(* Logix 5000 project; controller cal1615 1756-L62 rev 20.11; software revision 20.05; part 19 of 81 *)
(* tags used below, declared in another part *)
   FAULT : BOOL;   // Fault AFI
   HMI : BOOL;   // AFI HMI
   p01_param_oven_timer_presets : DINT[32];   // System Parameter Oven Timer Presets
   p01_param_process_air_hl : REAL;   // Machine Parameter Process Air High Limit
   p01_sys_lc : Limit_Clamp;   // Zone 1 Misc Control Limit Clamp
   p01r09_pb_global_reset : BOOL;   // System Modes PB: Global Fault Reset
   p01r11 : routine;   // System Timer Presets
   p02_real_from_hmi : hmi_real;   // MOP HMI Iface Real from HMI
   p11_dint_to_hmi : DINT[16];   // Zone 1 Temperature Control VFDs On
   p11_param_fast_to_soak : REAL;   // Zone 1 Parameter Fast to Soak Control
   p11_param_lfl_hhl : REAL;   // Zone 1 Parameter High High Lower Flash Limit
   p11_param_lfl_hl : REAL;   // Zone 1 Parameter High LFL Limit
   p11_param_pid1_ff : REAL;   // Zone 1 Parameter Fast PID Bias
   p11_param_pid1_kd : REAL;   // Zone 1 Parameter Fast PID Derivative Gain
   p11_param_pid1_ki : REAL;   // Zone 1 Parameter Fast PID Integral Gain
   p11_param_pid1_kp : REAL;   // Zone 1 Parameter Fast PID Proportional Gain
   p11_param_pid2_ff : REAL;   // Zone 1 Parameter Auto PID Bias
   p11_param_pid2_kd : REAL;   // Zone 1 Parameter Auto PID Derivative Gain
   p11_param_pid2_ki : REAL;   // Zone 1 Parameter Auto PID Integral Gain
   p11_param_pid2_kp : REAL;   // Zone 1 Parameter Auto PID Proportional Gain
   p11_param_shutdown_temp : REAL;   // Zone 1 Parameter Zone Shutdown Temperature
   p11_param_soak_to_fast : REAL;   // Zone 1 Parameter Soak to Fast Control
   p11_param_tc01_dev : REAL;   // Zone 1 Parameter Oven Temperature Deviation from Setpoint
   p11_param_tc01_hl : REAL;   // Zone 1 Parameter Process Air High Limit
   p11_param_tc01z : REAL;   // Zone 1 Parameter Process Temperature Zero Offset
   p11_param_tc02z : REAL;   // Zone 1 Parameter SupplyTemperature Zero Offset
   p11_param_zone_pressure : REAL;   // Zone 1 Parameter High Pressure LImit
   p11r01 : routine;   // Zone 1 Main
   p11r02 : routine;   // Zone 1 Misc Control
   p11r02_timer_warning : TIMER[4];   // Zone 1 Misc Control Warning Delay
   p11r07 : routine;   // Zone 1 Alarms
   p11r07_timer_fault : TIMER[4];   // Zone 1 Alarms Fault Delay
   p11r07_timer_warning : TIMER[4];   // Zone 1 Alarms Warning Delay
   p11r08 : routine;   // Zone 1 Warnings
   p11r08_timer_fault : TIMER[4];   // Zone 1 Warnings Fault Delay
   p11r08_timer_warning : TIMER[4];   // Zone 1 Warnings Warning Delay
   p11r09 : routine;   // Zone 1 Modes
   p11r09_timer_fault : TIMER[4];   // Zone 1 Modes Fault Delay
   p11r09_timer_warning : TIMER[8];   // Zone 1 Modes Warning Delay
   p11r10 : routine;   // Zone 1
   p11r20 : routine;   // Zone 1 Temp Sequence
   p11r30 : routine;   // Zone 1 Temperature Control
   p11r30_cv_man_sp : REAL;   // Zone 1 Temperature Control Manual Heat Control Valve Setpoint
   p11r30_temp_deviation_setpoint : DINT;
   p11r30_timer_fault : TIMER[16];   // Zone 1 Temperature Control Fault Delay
   p11r30_timer_warning : TIMER[12];   // Zone 1 Temperature Control Warning Delay
   p11r31 : routine;   // Zone 1 Exhaust VFD
   p11r31_timer_fault : TIMER[5];   // Zone 1 Exhaust VFD Fault Timer
   p11r31_timer_warning : TIMER[5];   // Zone 1 Exhaust VFD Waringing Timer
   p11r32 : routine;   // Zone 1 Recirc VFD
   p11r32_timer_fault : TIMER[5];   // Zone 1 Recirc VFD Fault Timer
   p11r32_timer_warning : TIMER[5];   // Zone 1 Supply VFD Warning Timer
(* P11_Zone_1, continued *)

ROUTINE R07_Alarms   (* ladder *)
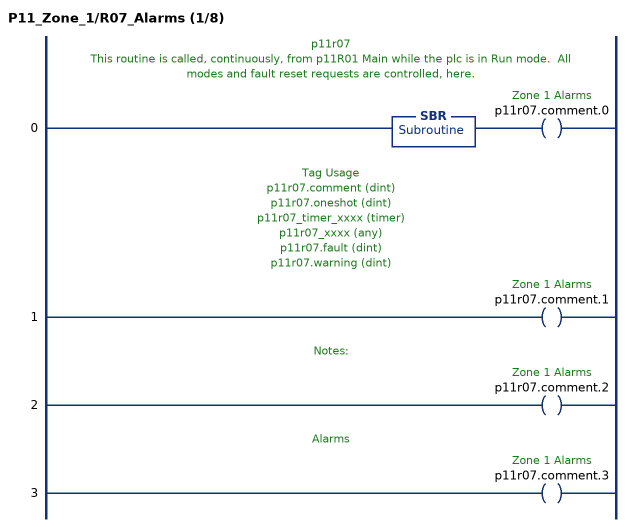
   // p11r07
   // This routine is called, continuously, from p11R01 Main while the plc is in Run mode.  All modes and fault reset requests are controlled, here.
   0: SBR()OTE(p11r07.comment.0);
   // Tag Usage
   // p11r07.comment (dint)
   // p11r07.oneshot (dint)
   // p11r07_timer_xxxx (timer)
   // p11r07_xxxx (any)
   // p11r07.fault (dint)
   // p11r07.warning (dint)
   1: OTE(p11r07.comment.1);
   // Notes:
   2: OTE(p11r07.comment.2);
   // Alarms
   3: OTE(p11r07.comment.3);
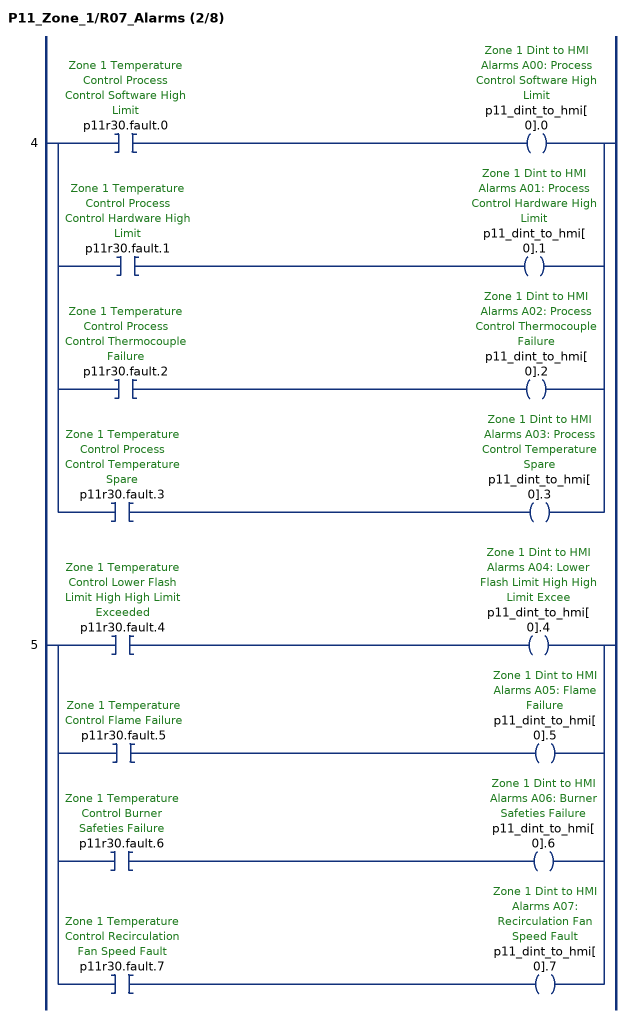
   4: [XIC(p11r30.fault.0) OTE(p11_dint_to_hmi[0].0) ,XIC(p11r30.fault.1) OTE(p11_dint_to_hmi[0].1) ,XIC(p11r30.fault.2) OTE(p11_dint_to_hmi[0].2) ,XIC(p11r30.fault.3) OTE(p11_dint_to_hmi[0].3) ];
   5: [XIC(p11r30.fault.4) OTE(p11_dint_to_hmi[0].4) ,XIC(p11r30.fault.5) OTE(p11_dint_to_hmi[0].5) ,XIC(p11r30.fault.6) OTE(p11_dint_to_hmi[0].6) ,XIC(p11r30.fault.7) OTE(p11_dint_to_hmi[0].7) ];
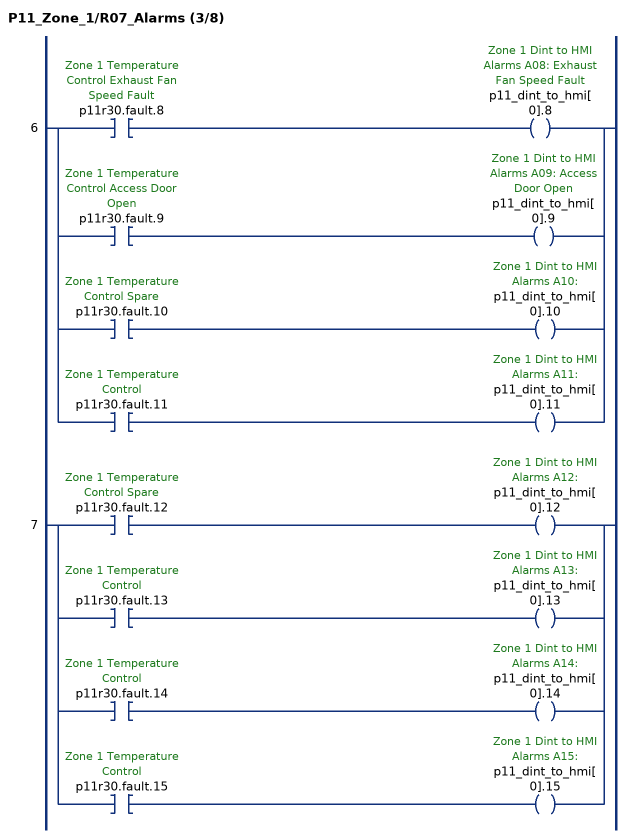
   6: [XIC(p11r30.fault.8) OTE(p11_dint_to_hmi[0].8) ,XIC(p11r30.fault.9) OTE(p11_dint_to_hmi[0].9) ,XIC(p11r30.fault.10) OTE(p11_dint_to_hmi[0].10) ,XIC(p11r30.fault.11) OTE(p11_dint_to_hmi[0].11) ];
   7: [XIC(p11r30.fault.12) OTE(p11_dint_to_hmi[0].12) ,XIC(p11r30.fault.13) OTE(p11_dint_to_hmi[0].13) ,XIC(p11r30.fault.14) OTE(p11_dint_to_hmi[0].14) ,XIC(p11r30.fault.15) OTE(p11_dint_to_hmi[0].15) ];
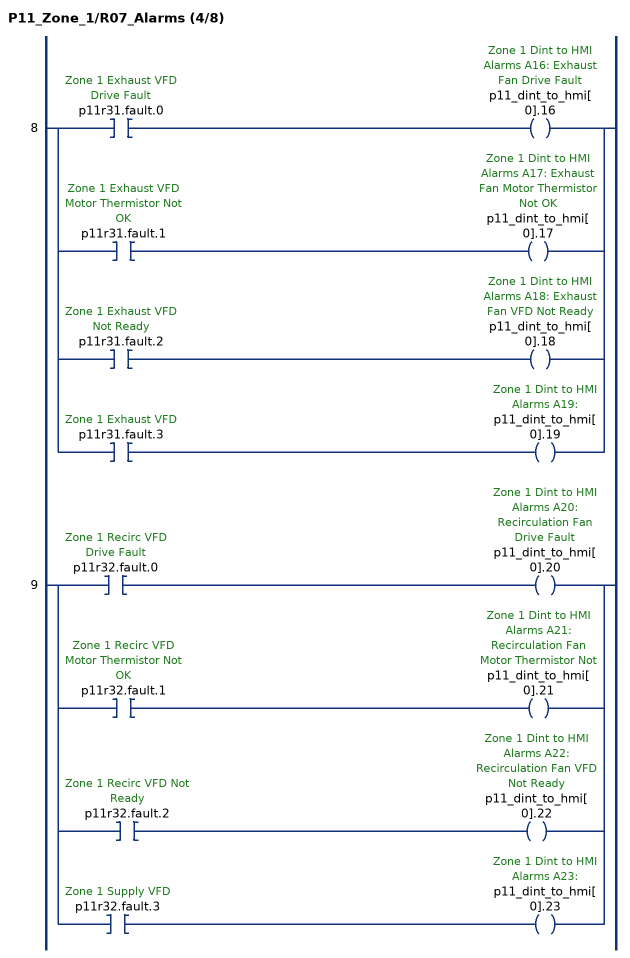
   8: [XIC(p11r31.fault.0) OTE(p11_dint_to_hmi[0].16) ,XIC(p11r31.fault.1) OTE(p11_dint_to_hmi[0].17) ,XIC(p11r31.fault.2) OTE(p11_dint_to_hmi[0].18) ,XIC(p11r31.fault.3) OTE(p11_dint_to_hmi[0].19) ];
   9: [XIC(p11r32.fault.0) OTE(p11_dint_to_hmi[0].20) ,XIC(p11r32.fault.1) OTE(p11_dint_to_hmi[0].21) ,XIC(p11r32.fault.2) OTE(p11_dint_to_hmi[0].22) ,XIC(p11r32.fault.3) OTE(p11_dint_to_hmi[0].23) ];
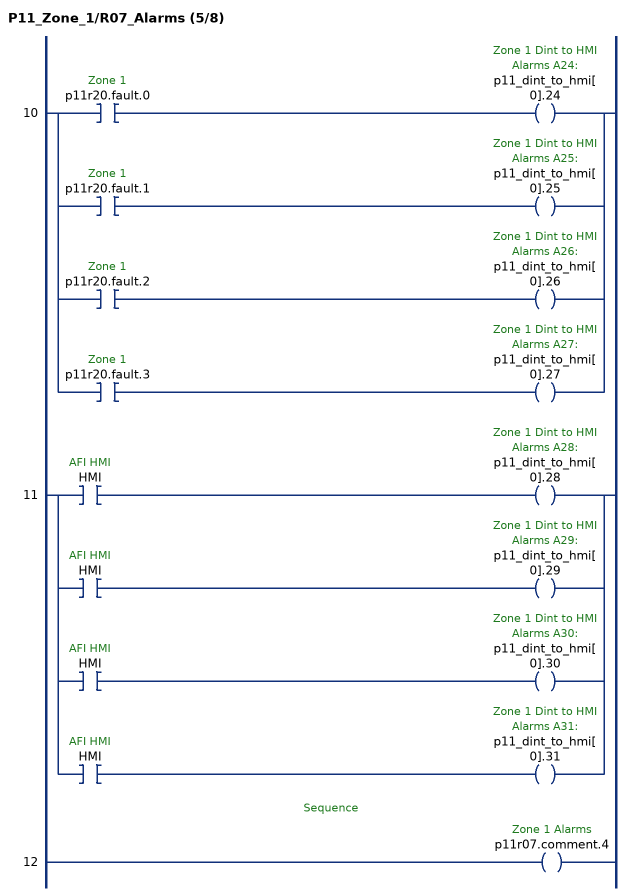
   10: [XIC(p11r20.fault.0) OTE(p11_dint_to_hmi[0].24) ,XIC(p11r20.fault.1) OTE(p11_dint_to_hmi[0].25) ,XIC(p11r20.fault.2) OTE(p11_dint_to_hmi[0].26) ,XIC(p11r20.fault.3) OTE(p11_dint_to_hmi[0].27) ];
   11: [XIC(HMI) OTE(p11_dint_to_hmi[0].28) ,XIC(HMI) OTE(p11_dint_to_hmi[0].29) ,XIC(HMI) OTE(p11_dint_to_hmi[0].30) ,XIC(HMI) OTE(p11_dint_to_hmi[0].31) ];
   // Sequence
   12: OTE(p11r07.comment.4);
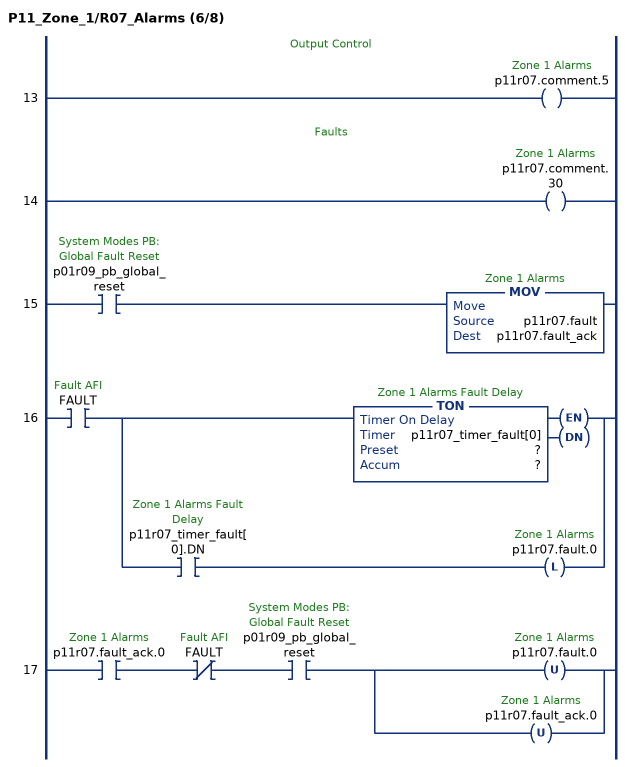
   // Output Control
   13: OTE(p11r07.comment.5);
   // Faults
   14: OTE(p11r07.comment.30);
   15: XIC(p01r09_pb_global_reset)MOV(p11r07.fault,p11r07.fault_ack);
   16: XIC(FAULT)[TON(p11r07_timer_fault[0],?,?) ,XIC(p11r07_timer_fault[0].DN) OTL(p11r07.fault.0) ];
   17: XIC(p11r07.fault_ack.0)XIO(FAULT)XIC(p01r09_pb_global_reset)[OTU(p11r07.fault.0) ,OTU(p11r07.fault_ack.0) ];
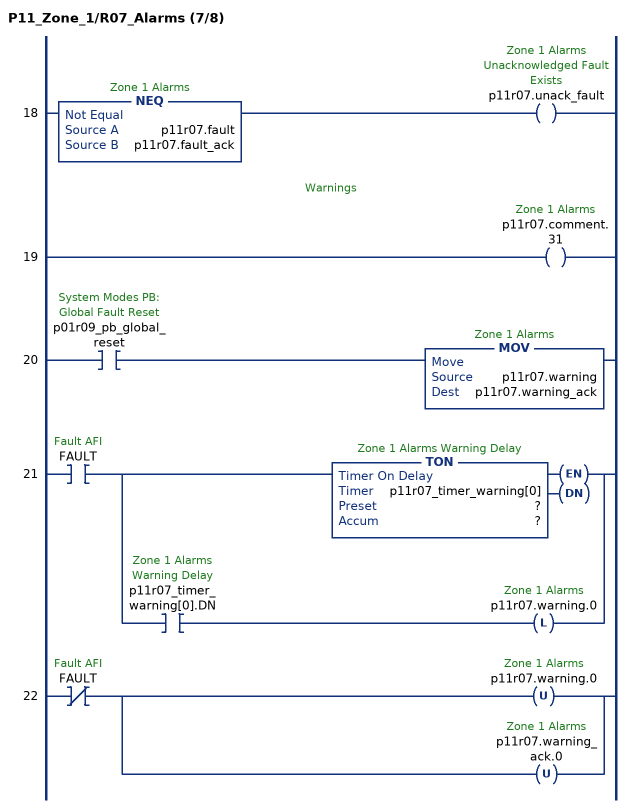
   18: NEQ(p11r07.fault,p11r07.fault_ack)OTE(p11r07.unack_fault);
   // Warnings
   19: OTE(p11r07.comment.31);
   20: XIC(p01r09_pb_global_reset)MOV(p11r07.warning,p11r07.warning_ack);
   21: XIC(FAULT)[TON(p11r07_timer_warning[0],?,?) ,XIC(p11r07_timer_warning[0].DN) OTL(p11r07.warning.0) ];
   22: XIO(FAULT)[OTU(p11r07.warning.0) ,OTU(p11r07.warning_ack.0) ];
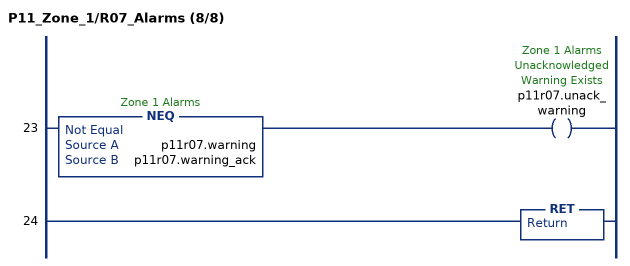
   23: NEQ(p11r07.warning,p11r07.warning_ack)OTE(p11r07.unack_warning);
   24: RET();
END_ROUTINE

ROUTINE R08_Warnings   (* ladder *)
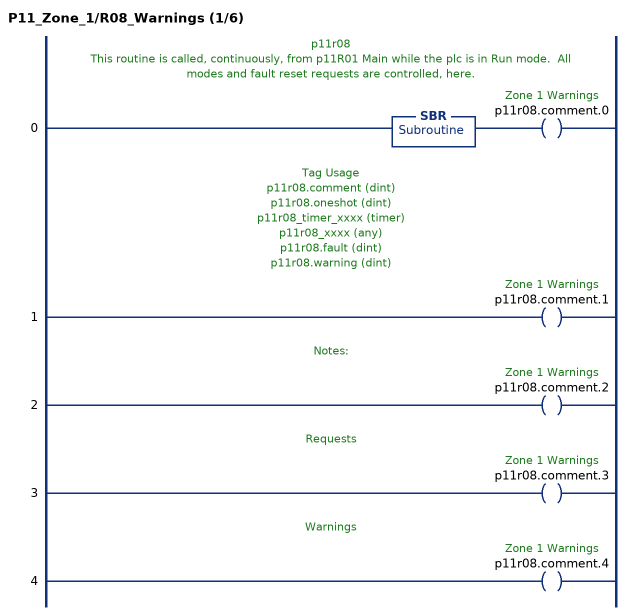
   // p11r08
   // This routine is called, continuously, from p11R01 Main while the plc is in Run mode.  All modes and fault reset requests are controlled, here.
   0: SBR()OTE(p11r08.comment.0);
   // Tag Usage
   // p11r08.comment (dint)
   // p11r08.oneshot (dint)
   // p11r08_timer_xxxx (timer)
   // p11r08_xxxx (any)
   // p11r08.fault (dint)
   // p11r08.warning (dint)
   1: OTE(p11r08.comment.1);
   // Notes:
   2: OTE(p11r08.comment.2);
   // Requests
   3: OTE(p11r08.comment.3);
   // Warnings
   4: OTE(p11r08.comment.4);
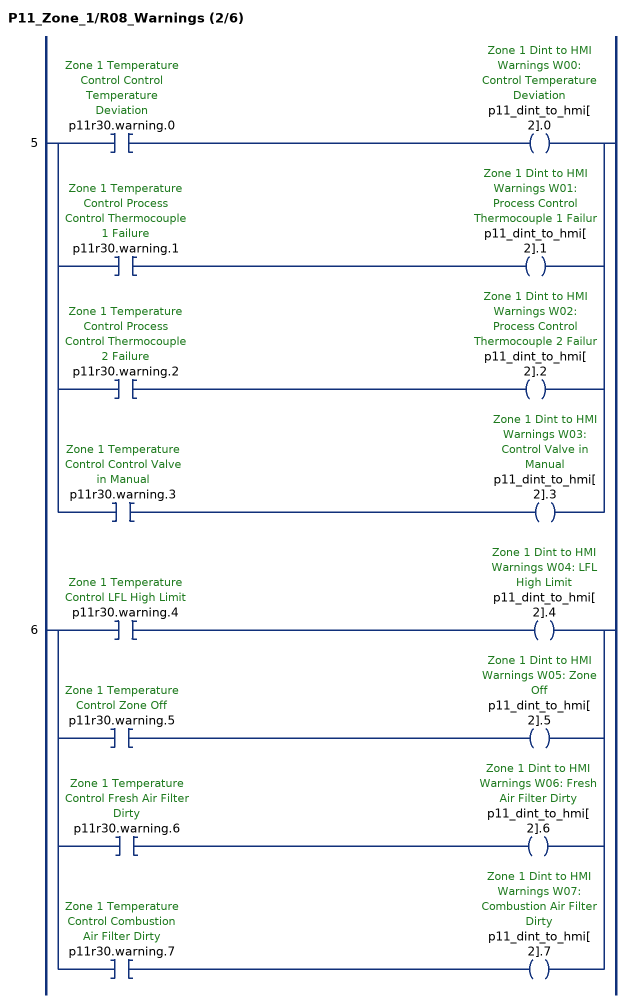
   5: [XIC(p11r30.warning.0) OTE(p11_dint_to_hmi[2].0) ,XIC(p11r30.warning.1) OTE(p11_dint_to_hmi[2].1) ,XIC(p11r30.warning.2) OTE(p11_dint_to_hmi[2].2) ,XIC(p11r30.warning.3) OTE(p11_dint_to_hmi[2].3) ];
   6: [XIC(p11r30.warning.4) OTE(p11_dint_to_hmi[2].4) ,XIC(p11r30.warning.5) OTE(p11_dint_to_hmi[2].5) ,XIC(p11r30.warning.6) OTE(p11_dint_to_hmi[2].6) ,XIC(p11r30.warning.7) OTE(p11_dint_to_hmi[2].7) ];
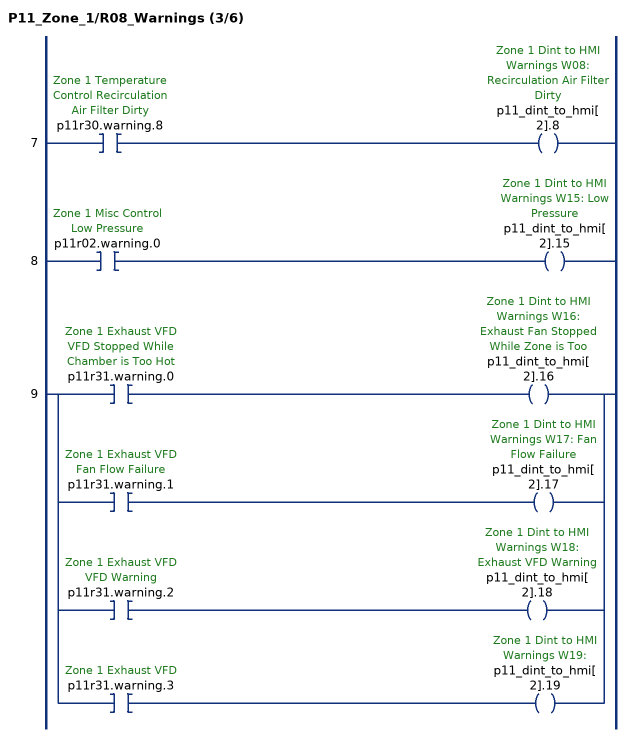
   7: XIC(p11r30.warning.8)OTE(p11_dint_to_hmi[2].8);
   8: XIC(p11r02.warning.0)OTE(p11_dint_to_hmi[2].15);
   9: [XIC(p11r31.warning.0) OTE(p11_dint_to_hmi[2].16) ,XIC(p11r31.warning.1) OTE(p11_dint_to_hmi[2].17) ,XIC(p11r31.warning.2) OTE(p11_dint_to_hmi[2].18) ,XIC(p11r31.warning.3) OTE(p11_dint_to_hmi[2].19) ];
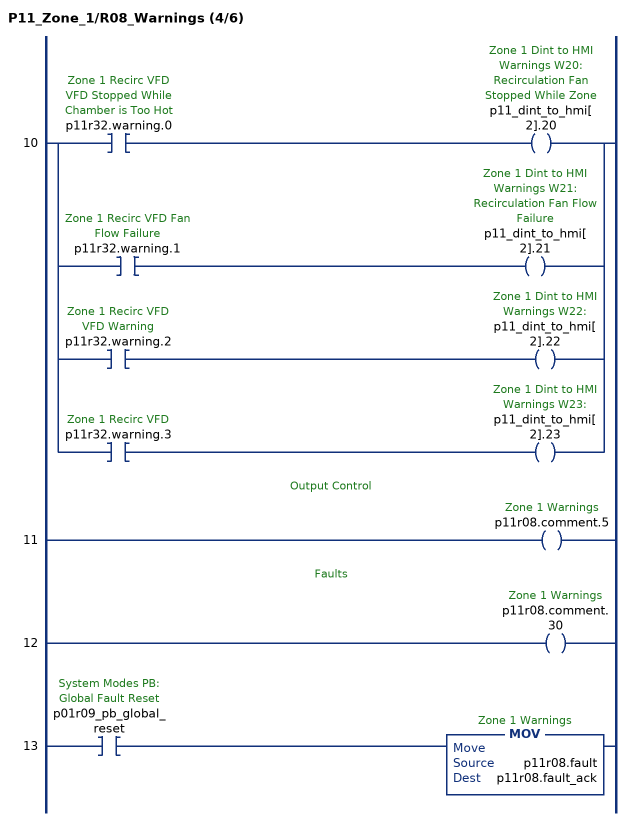
   10: [XIC(p11r32.warning.0) OTE(p11_dint_to_hmi[2].20) ,XIC(p11r32.warning.1) OTE(p11_dint_to_hmi[2].21) ,XIC(p11r32.warning.2) OTE(p11_dint_to_hmi[2].22) ,XIC(p11r32.warning.3) OTE(p11_dint_to_hmi[2].23) ];
   // Output Control
   11: OTE(p11r08.comment.5);
   // Faults
   12: OTE(p11r08.comment.30);
   13: XIC(p01r09_pb_global_reset)MOV(p11r08.fault,p11r08.fault_ack);
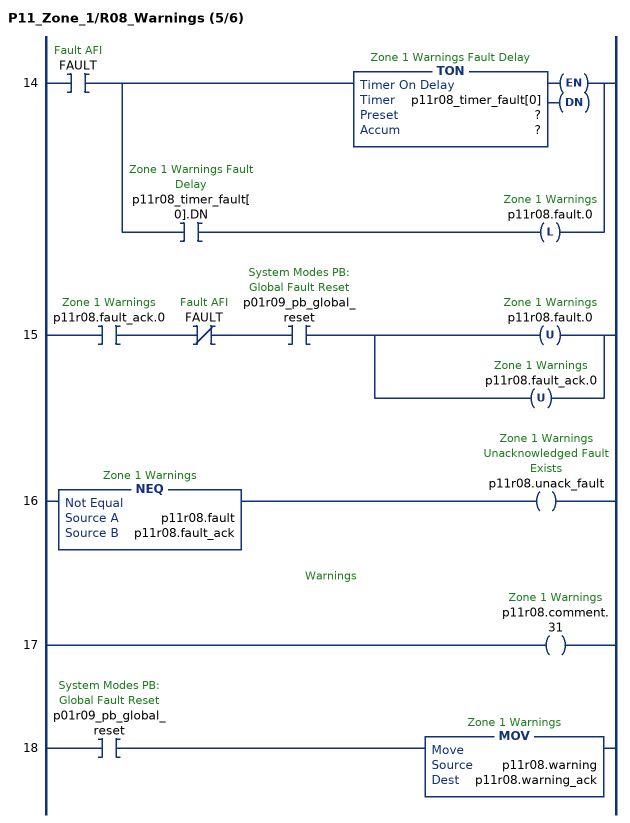
   14: XIC(FAULT)[TON(p11r08_timer_fault[0],?,?) ,XIC(p11r08_timer_fault[0].DN) OTL(p11r08.fault.0) ];
   15: XIC(p11r08.fault_ack.0)XIO(FAULT)XIC(p01r09_pb_global_reset)[OTU(p11r08.fault.0) ,OTU(p11r08.fault_ack.0) ];
   16: NEQ(p11r08.fault,p11r08.fault_ack)OTE(p11r08.unack_fault);
   // Warnings
   17: OTE(p11r08.comment.31);
   18: XIC(p01r09_pb_global_reset)MOV(p11r08.warning,p11r08.warning_ack);
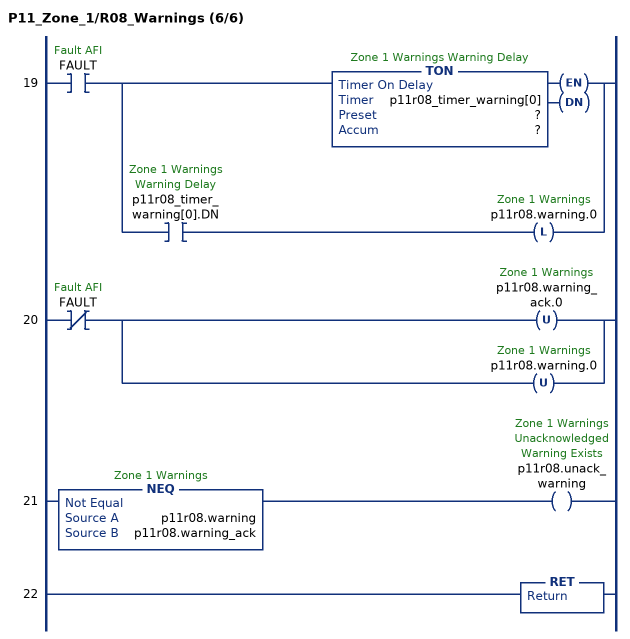
   19: XIC(FAULT)[TON(p11r08_timer_warning[0],?,?) ,XIC(p11r08_timer_warning[0].DN) OTL(p11r08.warning.0) ];
   20: XIO(FAULT)[OTU(p11r08.warning_ack.0) ,OTU(p11r08.warning.0) ];
   21: NEQ(p11r08.warning,p11r08.warning_ack)OTE(p11r08.unack_warning);
   22: RET();
END_ROUTINE

ROUTINE R09_Modes   (* ladder *)
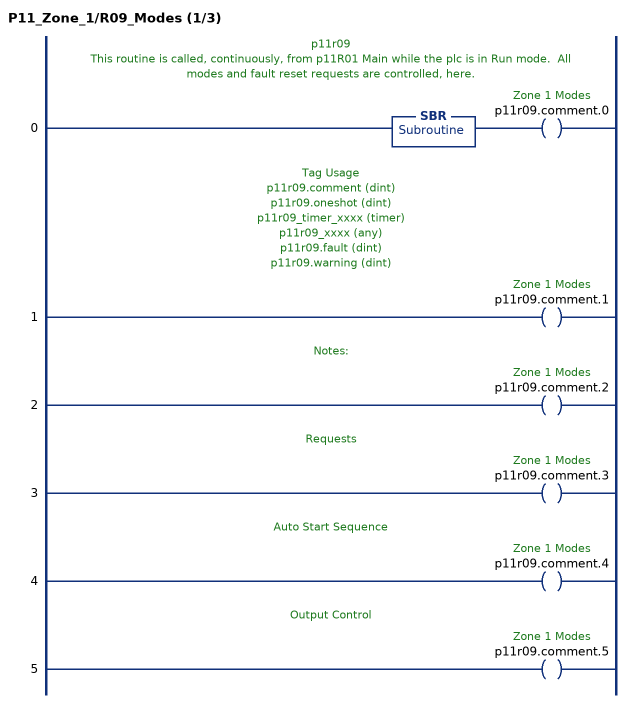
   // p11r09
   // This routine is called, continuously, from p11R01 Main while the plc is in Run mode.  All modes and fault reset requests are controlled, here.
   0: SBR()OTE(p11r09.comment.0);
   // Tag Usage
   // p11r09.comment (dint)
   // p11r09.oneshot (dint)
   // p11r09_timer_xxxx (timer)
   // p11r09_xxxx (any)
   // p11r09.fault (dint)
   // p11r09.warning (dint)
   1: OTE(p11r09.comment.1);
   // Notes:
   2: OTE(p11r09.comment.2);
   // Requests
   3: OTE(p11r09.comment.3);
   // Auto Start Sequence
   4: OTE(p11r09.comment.4);
   // Output Control
   5: OTE(p11r09.comment.5);
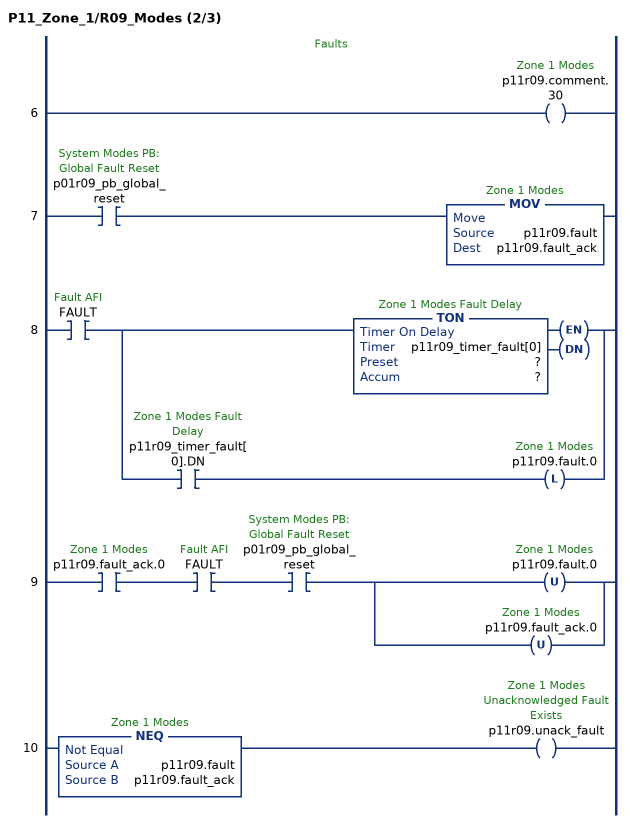
   // Faults
   6: OTE(p11r09.comment.30);
   7: XIC(p01r09_pb_global_reset)MOV(p11r09.fault,p11r09.fault_ack);
   8: XIC(FAULT)[TON(p11r09_timer_fault[0],?,?) ,XIC(p11r09_timer_fault[0].DN) OTL(p11r09.fault.0) ];
   9: XIC(p11r09.fault_ack.0)XIC(FAULT)XIC(p01r09_pb_global_reset)[OTU(p11r09.fault.0) ,OTU(p11r09.fault_ack.0) ];
   10: NEQ(p11r09.fault,p11r09.fault_ack)OTE(p11r09.unack_fault);
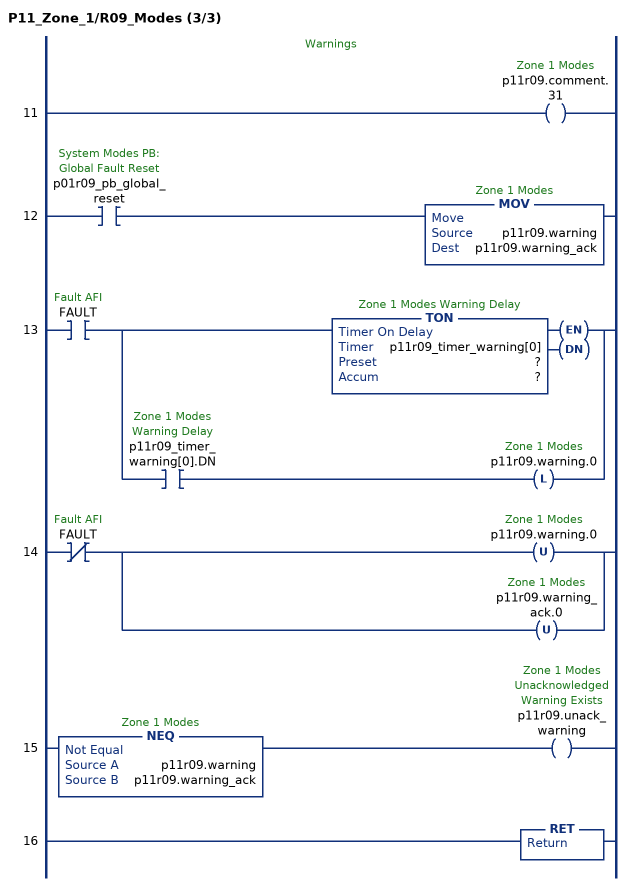
   // Warnings
   11: OTE(p11r09.comment.31);
   12: XIC(p01r09_pb_global_reset)MOV(p11r09.warning,p11r09.warning_ack);
   13: XIC(FAULT)[TON(p11r09_timer_warning[0],?,?) ,XIC(p11r09_timer_warning[0].DN) OTL(p11r09.warning.0) ];
   14: XIO(FAULT)[OTU(p11r09.warning.0) ,OTU(p11r09.warning_ack.0) ];
   15: NEQ(p11r09.warning,p11r09.warning_ack)OTE(p11r09.unack_warning);
   16: RET();
END_ROUTINE

ROUTINE R10_Parameters   (* ladder *)
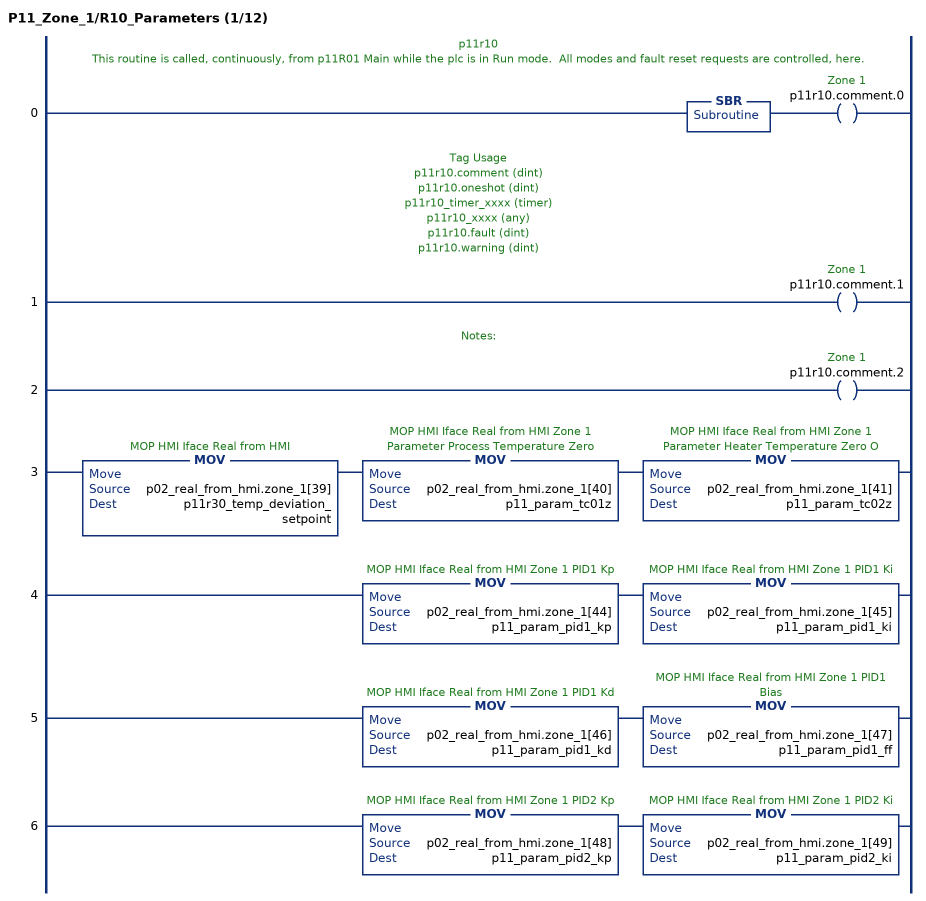
   // p11r10
   // This routine is called, continuously, from p11R01 Main while the plc is in Run mode.  All modes and fault reset requests are controlled, here.
   0: SBR()OTE(p11r10.comment.0);
   // Tag Usage
   // p11r10.comment (dint)
   // p11r10.oneshot (dint)
   // p11r10_timer_xxxx (timer)
   // p11r10_xxxx (any)
   // p11r10.fault (dint)
   // p11r10.warning (dint)
   1: OTE(p11r10.comment.1);
   // Notes:
   2: OTE(p11r10.comment.2);
   3: MOV(p02_real_from_hmi.zone_1[39],p11r30_temp_deviation_setpoint)MOV(p02_real_from_hmi.zone_1[40],p11_param_tc01z)MOV(p02_real_from_hmi.zone_1[41],p11_param_tc02z);
   4: MOV(p02_real_from_hmi.zone_1[44],p11_param_pid1_kp)MOV(p02_real_from_hmi.zone_1[45],p11_param_pid1_ki);
   5: MOV(p02_real_from_hmi.zone_1[46],p11_param_pid1_kd)MOV(p02_real_from_hmi.zone_1[47],p11_param_pid1_ff);
   6: MOV(p02_real_from_hmi.zone_1[48],p11_param_pid2_kp)MOV(p02_real_from_hmi.zone_1[49],p11_param_pid2_ki);
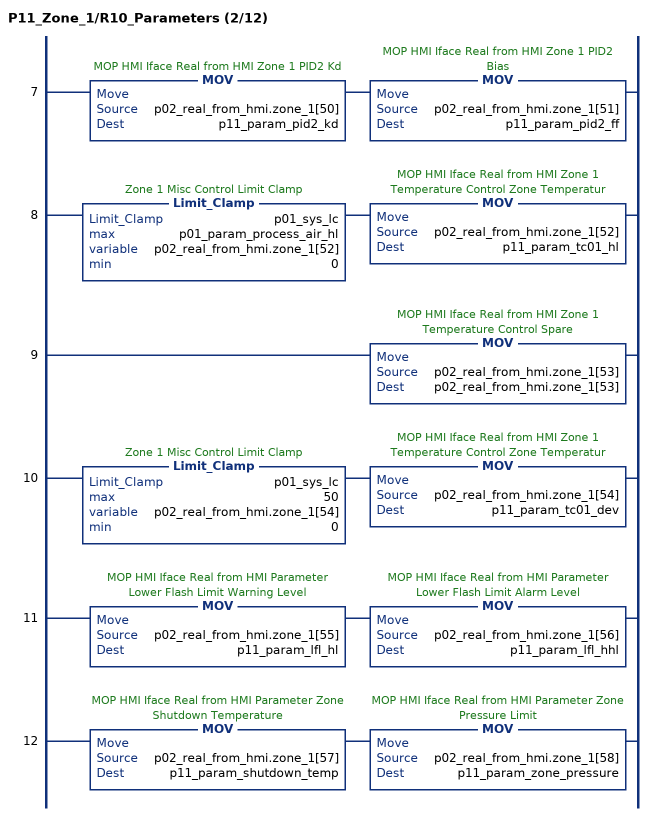
   7: MOV(p02_real_from_hmi.zone_1[50],p11_param_pid2_kd)MOV(p02_real_from_hmi.zone_1[51],p11_param_pid2_ff);
   8: Limit_Clamp(p01_sys_lc,p01_param_process_air_hl,p02_real_from_hmi.zone_1[52],0)MOV(p02_real_from_hmi.zone_1[52],p11_param_tc01_hl);
   9: MOV(p02_real_from_hmi.zone_1[53],p02_real_from_hmi.zone_1[53]);
   10: Limit_Clamp(p01_sys_lc,50,p02_real_from_hmi.zone_1[54],0)MOV(p02_real_from_hmi.zone_1[54],p11_param_tc01_dev);
   11: MOV(p02_real_from_hmi.zone_1[55],p11_param_lfl_hl)MOV(p02_real_from_hmi.zone_1[56],p11_param_lfl_hhl);
   12: MOV(p02_real_from_hmi.zone_1[57],p11_param_shutdown_temp)MOV(p02_real_from_hmi.zone_1[58],p11_param_zone_pressure);
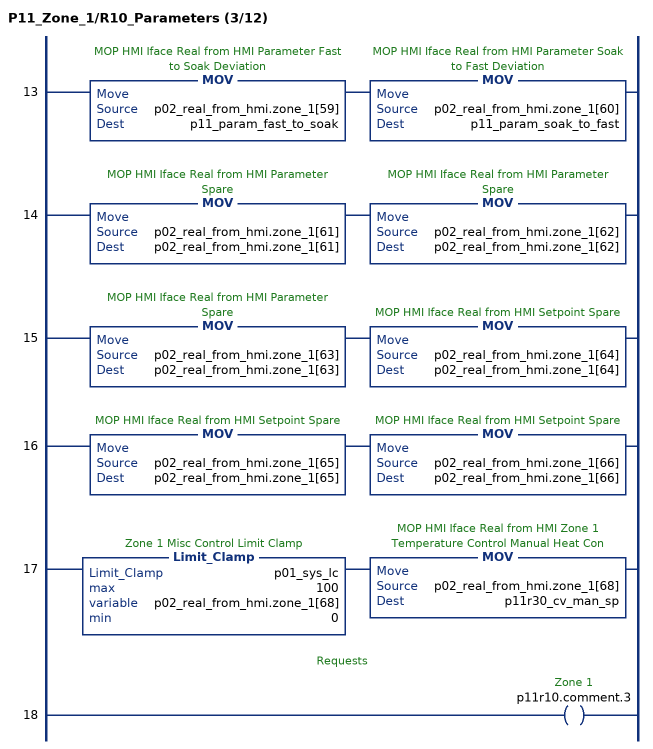
   13: MOV(p02_real_from_hmi.zone_1[59],p11_param_fast_to_soak)MOV(p02_real_from_hmi.zone_1[60],p11_param_soak_to_fast);
   14: MOV(p02_real_from_hmi.zone_1[61],p02_real_from_hmi.zone_1[61])MOV(p02_real_from_hmi.zone_1[62],p02_real_from_hmi.zone_1[62]);
   15: MOV(p02_real_from_hmi.zone_1[63],p02_real_from_hmi.zone_1[63])MOV(p02_real_from_hmi.zone_1[64],p02_real_from_hmi.zone_1[64]);
   16: MOV(p02_real_from_hmi.zone_1[65],p02_real_from_hmi.zone_1[65])MOV(p02_real_from_hmi.zone_1[66],p02_real_from_hmi.zone_1[66]);
   17: Limit_Clamp(p01_sys_lc,100,p02_real_from_hmi.zone_1[68],0)MOV(p02_real_from_hmi.zone_1[68],p11r30_cv_man_sp);
   // Requests
   18: OTE(p11r10.comment.3);
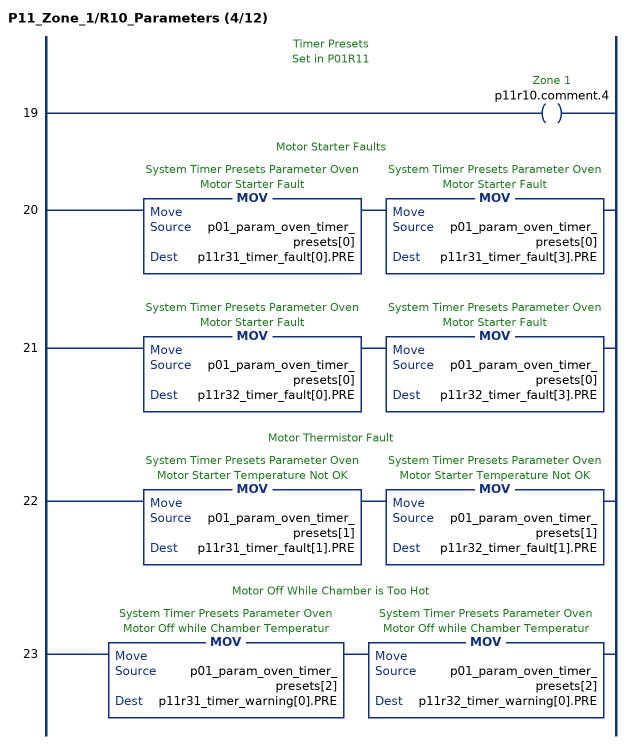
   // Timer Presets
   // Set in P01R11
   19: OTE(p11r10.comment.4);
   // Motor Starter Faults
   20: MOV(p01_param_oven_timer_presets[0],p11r31_timer_fault[0].PRE)MOV(p01_param_oven_timer_presets[0],p11r31_timer_fault[3].PRE);
   21: MOV(p01_param_oven_timer_presets[0],p11r32_timer_fault[0].PRE)MOV(p01_param_oven_timer_presets[0],p11r32_timer_fault[3].PRE);
   // Motor Thermistor Fault
   22: MOV(p01_param_oven_timer_presets[1],p11r31_timer_fault[1].PRE)MOV(p01_param_oven_timer_presets[1],p11r32_timer_fault[1].PRE);
   // Motor Off While Chamber is Too Hot
   23: MOV(p01_param_oven_timer_presets[2],p11r31_timer_warning[0].PRE)MOV(p01_param_oven_timer_presets[2],p11r32_timer_warning[0].PRE);
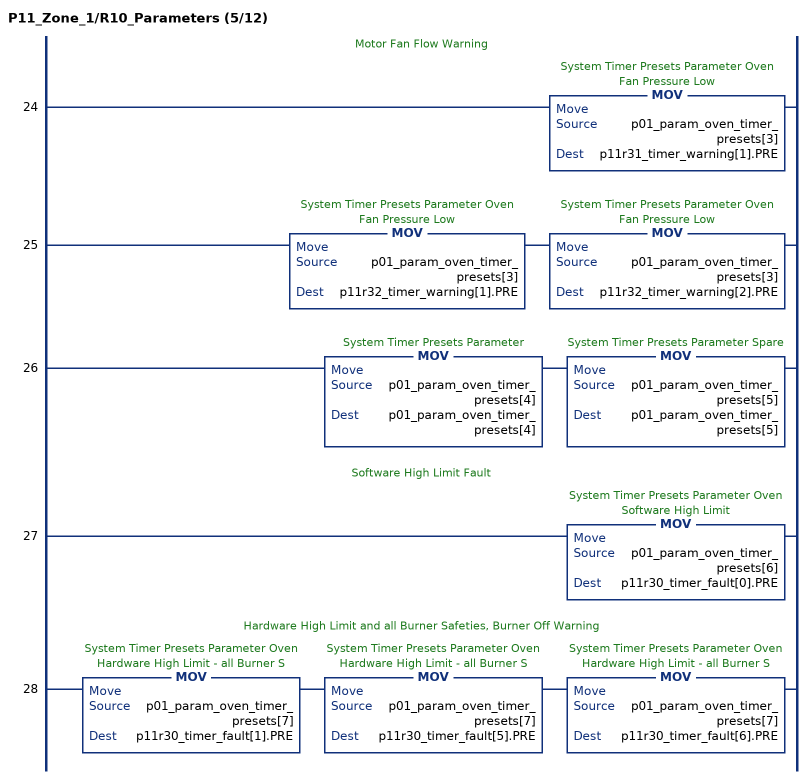
   // Motor Fan Flow Warning
   24: MOV(p01_param_oven_timer_presets[3],p11r31_timer_warning[1].PRE);
   25: MOV(p01_param_oven_timer_presets[3],p11r32_timer_warning[1].PRE)MOV(p01_param_oven_timer_presets[3],p11r32_timer_warning[2].PRE);
   26: MOV(p01_param_oven_timer_presets[4],p01_param_oven_timer_presets[4])MOV(p01_param_oven_timer_presets[5],p01_param_oven_timer_presets[5]);
   // Software High Limit Fault
   27: MOV(p01_param_oven_timer_presets[6],p11r30_timer_fault[0].PRE);
   // Hardware High Limit and all Burner Safeties, Burner Off Warning
   28: MOV(p01_param_oven_timer_presets[7],p11r30_timer_fault[1].PRE)MOV(p01_param_oven_timer_presets[7],p11r30_timer_fault[5].PRE)MOV(p01_param_oven_timer_presets[7],p11r30_timer_fault[6].PRE);
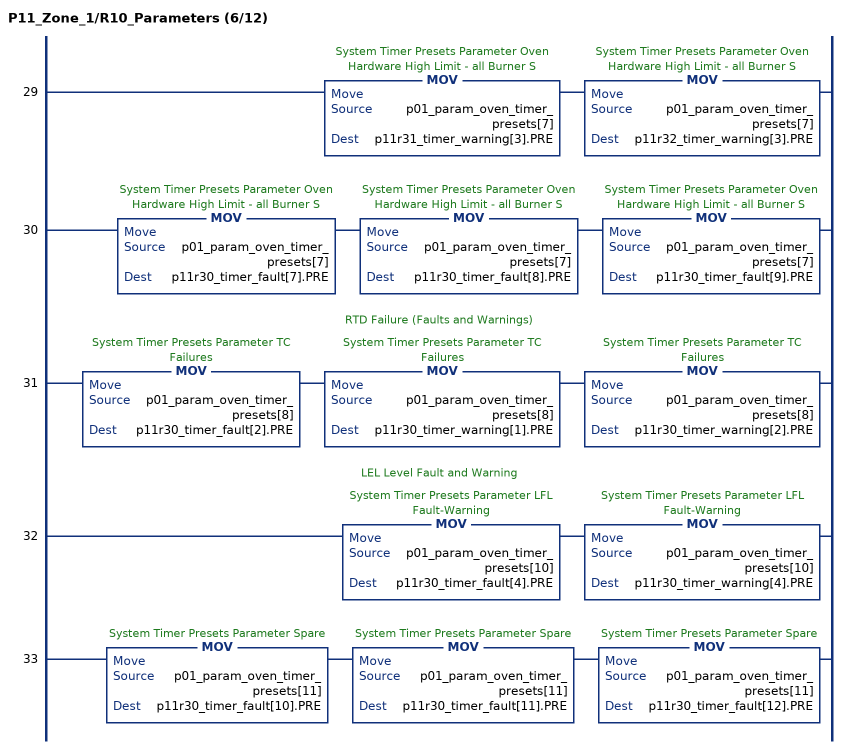
   29: MOV(p01_param_oven_timer_presets[7],p11r31_timer_warning[3].PRE)MOV(p01_param_oven_timer_presets[7],p11r32_timer_warning[3].PRE);
   30: MOV(p01_param_oven_timer_presets[7],p11r30_timer_fault[7].PRE)MOV(p01_param_oven_timer_presets[7],p11r30_timer_fault[8].PRE)MOV(p01_param_oven_timer_presets[7],p11r30_timer_fault[9].PRE);
   // RTD Failure (Faults and Warnings)
   31: MOV(p01_param_oven_timer_presets[8],p11r30_timer_fault[2].PRE)MOV(p01_param_oven_timer_presets[8],p11r30_timer_warning[1].PRE)MOV(p01_param_oven_timer_presets[8],p11r30_timer_warning[2].PRE);
   // LEL Level Fault and Warning
   32: MOV(p01_param_oven_timer_presets[10],p11r30_timer_fault[4].PRE)MOV(p01_param_oven_timer_presets[10],p11r30_timer_warning[4].PRE);
   33: MOV(p01_param_oven_timer_presets[11],p11r30_timer_fault[10].PRE)MOV(p01_param_oven_timer_presets[11],p11r30_timer_fault[11].PRE)MOV(p01_param_oven_timer_presets[11],p11r30_timer_fault[12].PRE);
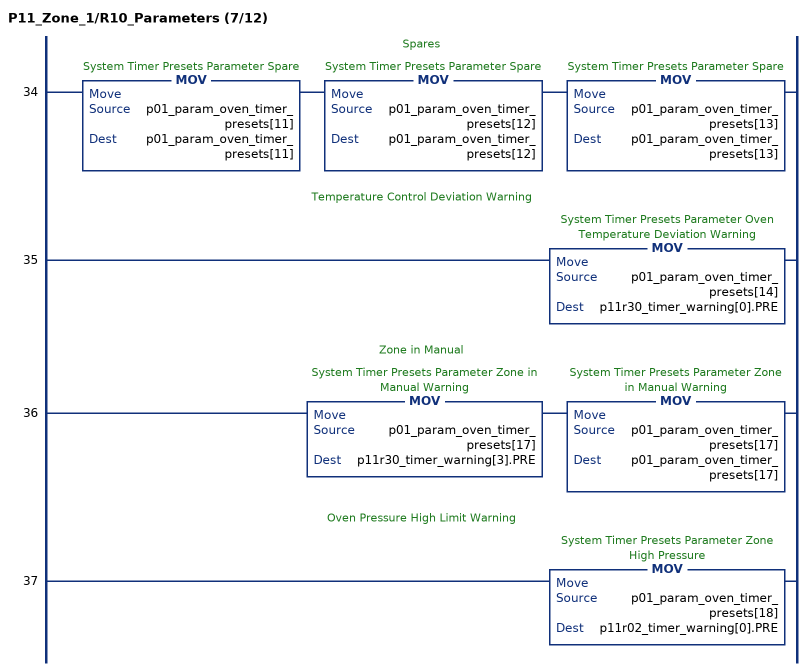
   // Spares
   34: MOV(p01_param_oven_timer_presets[11],p01_param_oven_timer_presets[11])MOV(p01_param_oven_timer_presets[12],p01_param_oven_timer_presets[12])MOV(p01_param_oven_timer_presets[13],p01_param_oven_timer_presets[13]);
   // Temperature Control Deviation Warning
   35: MOV(p01_param_oven_timer_presets[14],p11r30_timer_warning[0].PRE);
   // Zone in Manual
   36: MOV(p01_param_oven_timer_presets[17],p11r30_timer_warning[3].PRE)MOV(p01_param_oven_timer_presets[17],p01_param_oven_timer_presets[17]);
   // Oven Pressure High Limit Warning
   37: MOV(p01_param_oven_timer_presets[18],p11r02_timer_warning[0].PRE);
